Staubli VAL3: fhmns.pgx

public program fhmns(num x_nSec, string& x_sHMinSec[])
  local num l_nHour
  local num l_nMin
  local num l_nSec
begin
  //-----------------------------------------------------------------------
  //Header begin 开头
  //Description of program  程序描述
  //  Convert a num seconds in string hour : "xx h xx mn xx s".
  //  把时间的秒数转变成"xx h xx mn xx s"的形式
  //Input parameters  输入参数
  //  num x_nSec : 数值量x_nSec
  //    role : put a numerical expression that you want to convert in Hmns
  //    作用：放一个数值的表达式，这个表达式是你想去转换的
  //Output parameters  输出参数
  //  string x_sHMinSec :  字符串x_sHMinSec
  //    role : string hour correspond of your numerical expression
  //    作用：对应于你的数值表达式的字符串小时
  //Example
  //  call hmns(l_nSecond,l_sHMinSec)
  //
  //History
  //  Creation : 28-04-08 - f.Rob
  //Header end
  //-----------------------------------------------------------------------
  l_nHour=roundDown(x_nSec/3600)
  l_nMin=roundDown((x_nSec%3600)/60)
  l_nSec=roundDown(x_nSec-l_nHour*3600-l_nMin*60)
  x_sHMinSec=toString("3.0",l_nHour)+" h "+toString("2.0",l_nMin)+" mn "+toString("2.0",l_nSec)+" s"
end
